FUNCTION_BLOCK ALI_FIELDBUS_LINT_TO_SIGNAL (* Mirrors IN->OUT if Signal Valid. *)
  (* Standard: 61499-1 *)
  (* Version 1.0, 2026-05-31, franz *)
  PACKAGE logiBUS::signalprocessing::fieldbus;
  IMPORT signalprocessing::FIELDBUS_SIGNAL::NOT_AVAILABLE_DM;
  IMPORT signalprocessing::FIELDBUS_SIGNAL::VALID_SIGNAL_DW;
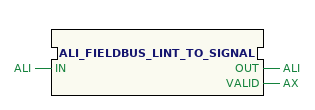
  SOCKETS
    IN : adapter::types::unidirectional::ALI; (* Input *)
  END_SOCKETS
  PLUGS
    OUT : adapter::types::unidirectional::ALI; (* Output Filtered *)
    VALID : adapter::types::unidirectional::AX; (* TRUE if Signal is VALID *)
  END_PLUGS
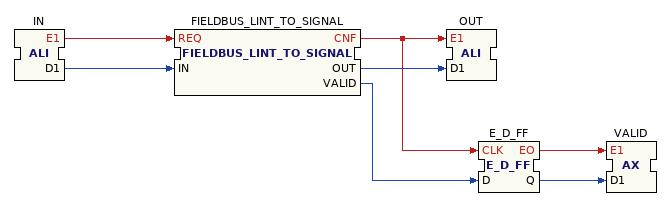
  FBS
    FIELDBUS_LINT_TO_SIGNAL : logiBUS::signalprocessing::fieldbus::FIELDBUS_LINT_TO_SIGNAL;
    E_D_FF : iec61499::events::E_D_FF;
  END_FBS
  EVENT_CONNECTIONS
    IN.E1 TO FIELDBUS_LINT_TO_SIGNAL.REQ;
    FIELDBUS_LINT_TO_SIGNAL.CNF TO OUT.E1;
    FIELDBUS_LINT_TO_SIGNAL.CNF TO E_D_FF.CLK;
    E_D_FF.EO TO VALID.E1;
  END_CONNECTIONS
  DATA_CONNECTIONS
    IN.D1 TO FIELDBUS_LINT_TO_SIGNAL.IN;
    FIELDBUS_LINT_TO_SIGNAL.OUT TO OUT.D1;
    FIELDBUS_LINT_TO_SIGNAL.VALID TO E_D_FF.D;
    E_D_FF.Q TO VALID.D1;
  END_CONNECTIONS
END_FUNCTION_BLOCK
